TYPE (* A Structure with 4 BOOLS *)
  (* Version 1.0, 2024-02-21, Franz Höpfinger, HR Agrartechnik GmbH *)
  ST04B : STRUCT
    B_00 : BOOL; (* BIT 00 *)
    B_01 : BOOL; (* BIT 01 *)
    B_02 : BOOL; (* BIT 02 *)
    B_03 : BOOL; (* BIT 03 *)
  END_STRUCT;
END_TYPE
